// TIA Portal V17 export
// export: Created 2026-01-01T00:00:00, ExportSetting WithDefaults, DisplayName synthetic-fixture, DisplayVersion machine-intelligence-v1.0.0
ORGANIZATION_BLOCK "OB1"   // OB, SCL
BEGIN

NETWORK
TITLE = 
FC_Mode();

NETWORK
TITLE = 
CV01Ctrl();

NETWORK
TITLE = 
CV02Ctrl();

NETWORK
TITLE = 
CV03Ctrl();

NETWORK
TITLE = 
CV04Ctrl();

NETWORK
TITLE = 
CV05Ctrl();

NETWORK
TITLE = 
CV06Ctrl();

NETWORK
TITLE = 
CV07Ctrl();

NETWORK
TITLE = 
CV08Ctrl();

NETWORK
TITLE = 
CV09Ctrl();

NETWORK
TITLE = 
CV10Ctrl();

NETWORK
TITLE = 
CV11Ctrl();

NETWORK
TITLE = 
CV12Ctrl();
END_ORGANIZATION_BLOCK
